(* IEC 61131-3 sources: rehub/fixtures/plc, 2 files *)

(* ---- boiler_approved.st ---- *)
(* Boiler temperature control *)
PROGRAM Boiler
VAR
    Setpoint : INT := 80;
    HighLimit : INT := 95;
END_VAR
IF Temp > Setpoint THEN
    Valve := FALSE;
END_IF;
END_PROGRAM

(* ---- boiler_updated.st ---- *)
(* Boiler temperature control *)
PROGRAM Boiler
VAR
    Setpoint : INT := 120;
    HighLimit : INT := 95;
    AdminPassword : STRING := 'hunter2';
END_VAR
IF Temp > Setpoint THEN
    Valve := FALSE;
END_IF;
TCON(REQ := TRUE, ADDR := '10.9.8.7');
SafetyInterlock := FALSE;
END_PROGRAM
